// TwinCAT 3 PLC project Untitled1
// ProgramVersion: 3.1.4022.7
// libraries:
//   Tc2_Standard, * (Beckhoff Automation GmbH)
//   Tc2_System, * (Beckhoff Automation GmbH)
//   Tc3_Module, * (Beckhoff Automation GmbH)
// project tree:
//   / PlcTask.TcTTO
//   POUs/ FBDelayCheck.TcPOU, MAIN.TcPOU
// real-time tasks:
//   TASK PlcTask: cycle T#10ms, priority 20, ADS port 350
// I/O:
//   DEVICE Device 1 (EtherCAT), AmsNetId 5.100.231.146.2.1
//     Term 1 (EK1200) [EK1200-5000 EtherCAT Power supply (2A E-Bus)]
//       Term 2 (EK1110) [EK1110 EtherCAT extension]
//     Term 3 (EK1100) [EK1100 EtherCAT Coupler (2A E-Bus)]
//       Term 4 (EL1809) [EL1809 16Ch. Dig. Input 24V, 3ms]
//       Term 5 (EL2809) [EL2809 16Ch. Dig. Output 24V, 0.5A]
//       Term 6 (EL3208) [EL3208 8Ch. Ana. Input PT100 (RTD)]
//       Term 7 (EL6731) [EL6731 PROFIBUS DP Master]
//       Term 8 (EL9011) [EL9011 End Terminal]
//   DEVICE Device 4 (COM Port)
//   DEVICE Device 2 (EL6731), AmsNetId 5.100.231.146.3.1

CONFIGURATION Untitled1
    RESOURCE PLC ON TwinCAT3
        TASK PlcTask(INTERVAL := T#10ms, PRIORITY := 20);
        PROGRAM MAIN WITH PlcTask : MAIN;
    END_RESOURCE
END_CONFIGURATION

// ---- POUs/MAIN.TcPOU
PROGRAM MAIN
VAR
	count1 :INT;
	F1 :FBDelayCheck;
END_VAR


F1(in := count1, delaytime := T#0.2S);

END_PROGRAM

// ---- POUs/FBDelayCheck.TcPOU
FUNCTION_BLOCK FBDelayCheck
VAR_INPUT
	in:INT;
	delaytime :TIME;  //T#0.2s
END_VAR

VAR_OUTPUT
	timeout_flag :BOOL;
	timeout_nums :INT;
END_VAR


VAR
	
	data1		:INT;
	fbRtrig 	:R_TRIG;
	fbTon 		:TON;
END_VAR


fbTon(IN:= (in = data1) ,PT:= delaytime);

fbRtrig(CLK:= fbTon.Q, Q=>timeout_flag);

IF timeout_flag THEN
	timeout_nums := timeout_nums+1;
END_IF

data1 :=in;

END_FUNCTION_BLOCK
